// TIA Portal V19 export
DATA_BLOCK "INPUT MAPPING DB"   // DB2
{ S7_Optimized_Access := 'FALSE' }
   VAR
      "EMERGENCY STOP" : Bool;
      "AIR FAIL" : Bool;
      HOOTER : Bool;
      "MGF FEED PUMP P-101 A MCB TRIP" : Bool;
      "MGF FEED PUMP P-101 B MCB TRIP" : Bool;
      "MGF BACK WASH  P-102 A MCB TRIP" : Bool;
      "MGF BACK WASH P-102 B MCB TRIP" : Bool;
      "UF FEED PUMP P-103 A MCB TRIP" : Bool;
      "UF FEED PUMP P-103 B MCB TRIP" : Bool;
      "UF BLOWER AB-201 A MCB TRIP" : Bool;
      "UF BLOWER AB-201 B MCB TRIP" : Bool;
      "UF BACKWASH P-201A TRIP" : Bool;
      "UF BACKWASH P-201B TRIP" : Bool;
      "FRL LOW" : Bool;
      SPARE_3 : Bool;
      SPARE_4 : Bool;
      "DM FEED PUMP P-502 A MPCB TRIP" : Bool;
      "DM FEED PUMP P-502 B MPCB TRIP" : Bool;
      "DM FEED PUMP P-502 C MPCB TRIP" : Bool;
      "CIP P-601" : Bool;
      "BACK WASH RECOVERY P-801 A MPCB TRIP" : Bool;
      "BACK WASH RECOVERY P-801 B MPCB TRIP" : Bool;
      "ABFV-101 FEED BACK OPEN FEED BACK" : Bool;
      "ABFV-101 FEED BACK CLOSE FEED BACK" : Bool;
      "ABFV-102 FEED BACK OPEN FEED BACK" : Bool;
      "ABFV-102 FEED BACK CLOSE FEED BACK" : Bool;
      "ABFV-103 FEED BACK OPEN FEED BACK" : Bool;
      "ABFV-103 FEED BACK CLOSE FEED BACK" : Bool;
      "ABFV-104 FEED BACK OPEN FEED BACK" : Bool;
      "ABFV-104 FEED BACK CLOSE FEED BACK" : Bool;
      "ABFV 105 FEED BACK OPEN" : Bool;
      "ABFV 105 FEED BACK CLOSE" : Bool;
      "ABV 201 FEED BACK OPEN" : Bool;
      "ABV 201 FEED BACK CLOSE" : Bool;
      "ABFV 201 FEED BACK OPEN" : Bool;
      "ABFV 201 FEED BACK CLOSE" : Bool;
      "ABFV 202 FEED BACK OPEN" : Bool;
      "ABFV 202 FEED BACK CLOSE" : Bool;
      "ABFV 203 FEED BACK OPEN" : Bool;
      "ABFV 203 FEED BACK CLOSE" : Bool;
      "ABFV 204 FEED BACK OPEN" : Bool;
      "ABFV 204 FEED BACK CLOSE" : Bool;
      "ABFV 205 FEED BACK OPEN" : Bool;
      "ABFV 205 FEED BACK CLOSE" : Bool;
      "ABFV 206 FEED BACK OPEN" : Bool;
      "ABFV 206 FEED BACK CLOSE" : Bool;
      "ABFV-207 FEED BACK OPEN" : Bool;
      "ABFV-207 FEED BACK CLOSE" : Bool;
      "ABFV-208 FEED BACK OPEN" : Bool;
      "ABFV-208 FEED BACK CLOSE" : Bool;
      "P-101 A MGF FEED PUMP" : Bool;
      "P-101 B MGF FEED PUMP" : Bool;
      "P-102 A MGF BACK WASH" : Bool;
      "P-102 B MGF BACK WASH" : Bool;
      "P-103 A UF FEED PUMP" : Bool;
      "P-103 B UF FEED PUMP" : Bool;
      "AB-201 A UF BLOWER" : Bool;
      "AB-201 B UF BLOWER" : Bool;
      "P-201 A UF BACK WASH" : Bool;
      "P-201 B UF BACK WASH" : Bool;
      "P-502 A DM FEED PUMP" : Bool;
      "P-502 B DM FEED PUMP" : Bool;
      "P-502 C ON" : Bool;
      "P-601 ON" : Bool;
      "P-801 A BACK WASH WAST FEED BACK" : Bool;
      "P-801 B BACK WASH WAST FEED BACK" : Bool;
      "SPARE(5)" : Bool;
      "SPARE(6)" : Bool;
      "SPARE(7)" : Bool;
      "SPARE(8)" : Bool;
      "SPARE(9)" : Bool;
      "SPARE(10)" : Bool;
      "ABFV 501 OPEN FEED BACK" : Bool;
      "ABFV 501 CLOSE FEED BACK" : Bool;
      "ABFV 502 OPEN FEED BACK" : Bool;
      "ABFV 502 CLOSE FEED BACK" : Bool;
      "PS 201 UF" : Bool;
      "SPARE(12)" : Bool;
   END_VAR
BEGIN
END_DATA_BLOCK
